(* IEC 61131-3 sources: Lasal/CPU_5344_V01/Class/IOLinkCommChecker, 1 file *)

(* ---- IOLinkCommChecker.st ---- *)
(*!
<Class
	Name               = "IOLinkCommChecker"
	Revision           = "0.0"
	RealtimeTask       = "false"
	CyclicTask         = "true"
	DefCyclictime      = "10 ms"
	BackgroundTask     = "false"
	Sigmatek           = "false"
	OSInterface        = "false"
	HighPriority       = "false"
	Automatic          = "false"
	UpdateMode         = "Prescan"
	SharedCommandTable = "true"
	Objectsize         = "(540,900)">
	<Channels>
		<Server Name="ClassSvr" Visualized="false" Initialize="false" WriteProtected="true" Retentive="false"/>
		<Server Name="CommOk" Visualized="false" Initialize="false" WriteProtected="true" Retentive="false"/>
		<Client Name="ioLinkObject1" Required="false" Internal="false"/>
		<Client Name="ioLinkObject10" Required="false" Internal="false"/>
		<Client Name="ioLinkObject11" Required="false" Internal="false"/>
		<Client Name="ioLinkObject12" Required="false" Internal="false"/>
		<Client Name="ioLinkObject13" Required="false" Internal="false"/>
		<Client Name="ioLinkObject14" Required="false" Internal="false"/>
		<Client Name="ioLinkObject15" Required="false" Internal="false"/>
		<Client Name="ioLinkObject2" Required="false" Internal="false"/>
		<Client Name="ioLinkObject3" Required="false" Internal="false"/>
		<Client Name="ioLinkObject4" Required="false" Internal="false"/>
		<Client Name="ioLinkObject5" Required="false" Internal="false"/>
		<Client Name="ioLinkObject6" Required="false" Internal="false"/>
		<Client Name="ioLinkObject7" Required="false" Internal="false"/>
		<Client Name="ioLinkObject8" Required="false" Internal="false"/>
		<Client Name="ioLinkObject9" Required="false" Internal="false"/>
	</Channels>
</Class>
*)
IOLinkCommChecker : CLASS
  //Servers:
	ClassSvr 	: SvrChCmd_DINT;
	CommOk 	: SvrCh_DINT;
  //Clients:
	ioLinkObject1 	: CltChCmd_SDCIDevice;
	ioLinkObject2 	: CltChCmd_SDCIDevice;
	ioLinkObject3 	: CltChCmd_SDCIDevice;
	ioLinkObject4 	: CltChCmd_SDCIDevice;
	ioLinkObject5 	: CltChCmd_SDCIDevice;
	ioLinkObject6 	: CltChCmd_SDCIDevice;
	ioLinkObject7 	: CltChCmd_SDCIDevice;
	ioLinkObject8 	: CltChCmd_SDCIDevice;
	ioLinkObject9 	: CltChCmd_SDCIDevice;
	ioLinkObject10 	: CltChCmd_SDCIDevice;
	ioLinkObject11 	: CltChCmd_SDCIDevice;
	ioLinkObject12 	: CltChCmd_SDCIDevice;
	ioLinkObject13 	: CltChCmd_SDCIDevice;
	ioLinkObject14 	: CltChCmd_SDCIDevice;
	ioLinkObject15 	: CltChCmd_SDCIDevice;
  //Variables:
		con1Ok 	: DINT;
		con2Ok 	: DINT;
		con3Ok 	: DINT;
		con4Ok 	: DINT;
		con5Ok 	: DINT;
		con6Ok 	: DINT;
		con7Ok 	: DINT;
		con8Ok 	: DINT;
		con9Ok 	: DINT;
		con10Ok 	: DINT;
		con11Ok 	: DINT;
		con12Ok 	: DINT;
		con13Ok 	: DINT;
		con14Ok 	: DINT;
		con15Ok 	: DINT;
  //Functions:

	FUNCTION VIRTUAL GLOBAL Init;

	FUNCTION VIRTUAL GLOBAL CyWork
		VAR_INPUT
			EAX 	: UDINT;
		END_VAR
		VAR_OUTPUT
			state (EAX) 	: UDINT;
		END_VAR;

	FUNCTION GLOBAL Prescan;
  //Tables:
	FUNCTION @STD
		VAR_OUTPUT
			ret_code	: CONFSTATES;
		END_VAR;
	FUNCTION GLOBAL TAB @CT_;
END_CLASS;

#pragma usingLtd SDCIDevice

FUNCTION VIRTUAL GLOBAL IOLinkCommChecker::Init
con1Ok := IsClientConnected(#ioLinkObject1);
con2Ok := IsClientConnected(#ioLinkObject2);
con3Ok := IsClientConnected(#ioLinkObject3);
con4Ok := IsClientConnected(#ioLinkObject4);
con5Ok := IsClientConnected(#ioLinkObject5);
con6Ok := IsClientConnected(#ioLinkObject6);
con7Ok := IsClientConnected(#ioLinkObject7);
con8Ok := IsClientConnected(#ioLinkObject8);
con9Ok := IsClientConnected(#ioLinkObject9);
con10Ok := IsClientConnected(#ioLinkObject10);
con11Ok := IsClientConnected(#ioLinkObject11);
con12Ok := IsClientConnected(#ioLinkObject12);
con13Ok := IsClientConnected(#ioLinkObject13);
con14Ok := IsClientConnected(#ioLinkObject14);
con15Ok := IsClientConnected(#ioLinkObject15);

END_FUNCTION

FUNCTION VIRTUAL GLOBAL IOLinkCommChecker::CyWork
	VAR_INPUT
		EAX 	: UDINT;
	END_VAR
	VAR_OUTPUT
		state (EAX) 	: UDINT;
	END_VAR

  //update vals
  Prescan();

  // check for each object if the state is classok. if not all ok, communication is lost.
  // one of the reasons for losing communication can be that cables are damaged or 24v too low

  if (con1Ok = 0 | ioLinkObject1 = _ClassOk) & // not connected or status is ok
     (con2Ok = 0 | ioLinkObject2 = _ClassOk) &
     (con3Ok = 0 | ioLinkObject3 = _ClassOk) &
     (con4Ok = 0 | ioLinkObject4 = _ClassOk) &
     (con5Ok = 0 | ioLinkObject5 = _ClassOk) &
     (con6Ok = 0 | ioLinkObject6 = _ClassOk) &
     (con7Ok = 0 | ioLinkObject7 = _ClassOk) &
     (con8Ok = 0 | ioLinkObject8 = _ClassOk) &
     (con9Ok = 0 | ioLinkObject9 = _ClassOk) &
     (con10Ok = 0 | ioLinkObject10 = _ClassOk) &
     (con11Ok = 0 | ioLinkObject11 = _ClassOk) &
     (con12Ok = 0 | ioLinkObject12 = _ClassOk) &
     (con13Ok = 0 | ioLinkObject13 = _ClassOk) &
     (con14Ok = 0 | ioLinkObject14 = _ClassOk) &
     (con15Ok = 0 | ioLinkObject15 = _ClassOk)
  then
    CommOk := 1;
  else
    CommOk := 0;
  end_if;

	state := READY;

END_FUNCTION

FUNCTION GLOBAL IOLinkCommChecker::Prescan
if con1Ok then ioLinkObject1 := ioLinkObject1.Read(); end_if;
if con2Ok then ioLinkObject2 := ioLinkObject2.Read(); end_if;
if con3Ok then ioLinkObject3 := ioLinkObject3.Read(); end_if;
if con4Ok then ioLinkObject4 := ioLinkObject4.Read(); end_if;
if con5Ok then ioLinkObject5 := ioLinkObject5.Read(); end_if;
if con6Ok then ioLinkObject6 := ioLinkObject6.Read(); end_if;
if con7Ok then ioLinkObject7 := ioLinkObject7.Read(); end_if;
if con8Ok then ioLinkObject8 := ioLinkObject8.Read(); end_if;
if con9Ok then ioLinkObject9 := ioLinkObject9.Read(); end_if;
if con10Ok then ioLinkObject10 := ioLinkObject10.Read(); end_if;
if con11Ok then ioLinkObject11 := ioLinkObject11.Read(); end_if;
if con12Ok then ioLinkObject12 := ioLinkObject12.Read(); end_if;
if con13Ok then ioLinkObject13 := ioLinkObject13.Read(); end_if;
if con14Ok then ioLinkObject14 := ioLinkObject14.Read(); end_if;
if con15Ok then ioLinkObject15 := ioLinkObject15.Read(); end_if;
END_FUNCTION
